Omron Sysmac Studio project ARY_SearchMinMax (Sysmac Studio 1.65.0.64007, StandardProject)

# Controller new_Controller_0: NX1P2-1040DT1 version 1.69
Task PrimaryTask (priority 4, period or condition 2000): Program0

VAR_GLOBAL RETAIN
    Alarm : ARRAY[0..250] OF BOOL;  (* published *)
END_VAR
VAR_GLOBAL
    IN_Motor1_Ariza : BOOL;
    IN_Motor2_Ariza : BOOL;
    IN_Motor3_Ariza : BOOL;
    IN_Motor4_Ariza : BOOL;
    IN_Motor5_Ariza : BOOL;
    InoutPos : UINT;
    Alarm_Var : BOOL;
    Alarm_Sayisi : UINT;
END_VAR

PROGRAM Program0
VAR_EXTERNAL
    IN_Motor1_Ariza : BOOL;
    Alarm : ARRAY[0..250] OF BOOL;
    IN_Motor2_Ariza : BOOL;
    IN_Motor3_Ariza : BOOL;
    IN_Motor4_Ariza : BOOL;
    IN_Motor5_Ariza : BOOL;
    InoutPos : UINT;
    Alarm_Var : BOOL;
    Alarm_Sayisi : UINT;
END_VAR

(* Section ArySearch_Kullanimi: ladder, written here as Structured Text *)

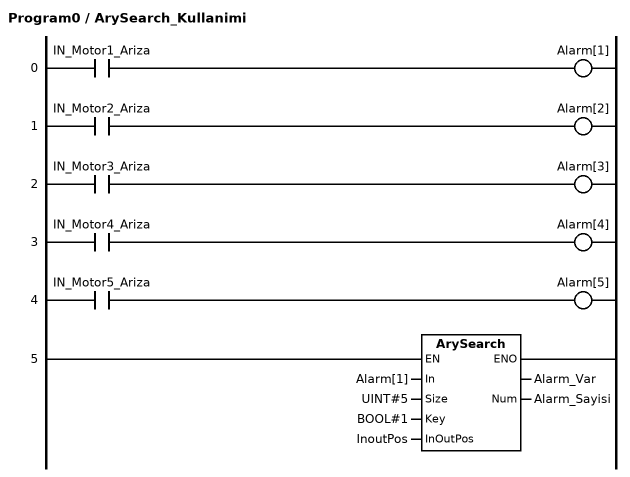
(* Rung 0 *)
Alarm[1] := IN_Motor1_Ariza;
(* Rung 1 *)
Alarm[2] := IN_Motor2_Ariza;
(* Rung 2 *)
Alarm[3] := IN_Motor3_Ariza;
(* Rung 3 *)
Alarm[4] := IN_Motor4_Ariza;
(* Rung 4 *)
Alarm[5] := IN_Motor5_Ariza;
(* Rung 5 *)
Alarm_Var := ArySearch(In := Alarm[1], Size := UINT#5, Key := BOOL#1, InOutPos := InoutPos, Num => Alarm_Sayisi);
END_PROGRAM